// TIA Portal V21 export
FUNCTION_BLOCK "FB610"   // FB610, LAD
TITLE = FB610
{ S7_Optimized_Access := 'FALSE' }
AUTHOR : PRECISE
FAMILY : PRECISE
// CIP SYSTEM DRAIN
// stored: AutoNumber false, SetENOAutomatically false
   VAR_INPUT
      CycleEnable : Bool;
      CycleRunning : Bool;
      SecPulse : Bool;
      AlwaysTrue : Bool;
      SetTime : Int := 30;
      Loops : Int;
      DelayBetweenLoops : Int := 3;
   END_VAR
   VAR_OUTPUT
      Started : Bool;
      ParaOut : "SystemDrainOutputs";
      TimePv : DInt;
      StepStatus : String[60];
   END_VAR
   VAR_IN_OUT
      Over : Bool;
      OverTemp : Bool;
      Popup : Bool;
      PopupAck : Bool;
      PopUpSel : Bool;
   END_VAR
   VAR
      RE1 : Bool;
      "Timer" { S7_SetPoint := 'True'} : "FB101";
   END_VAR
   VAR_TEMP   // added for the SCL form of the ladder/FBD networks
      _w1 : Bool;
      _w2 : Bool;
      _w3 : Bool;
   END_VAR
BEGIN

REGION Network 1: SystemDrainStarted
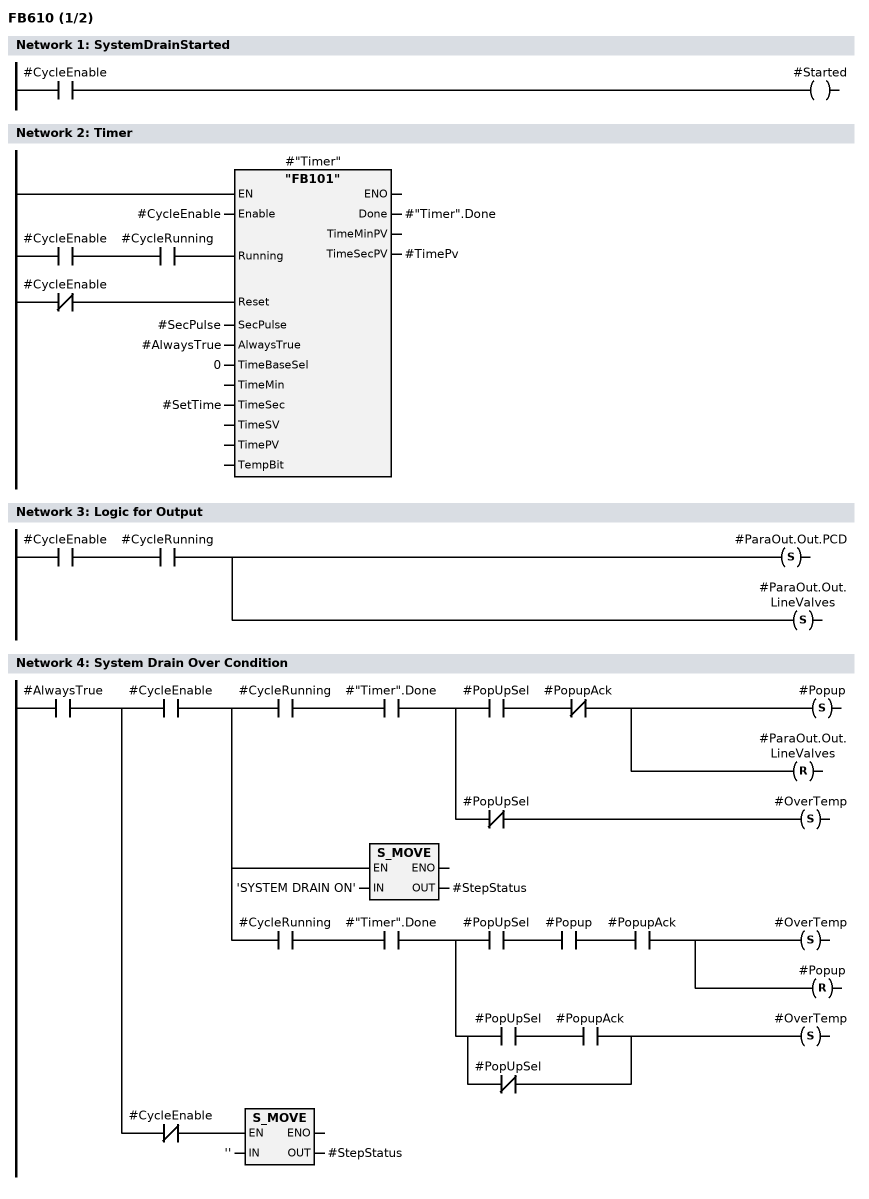
   RUNG wire#powerrail
      Contact( #CycleEnable )
      Coil( #Started )
   END_RUNG
   // the same network as SCL:
   #Started := #CycleEnable;
END_REGION

REGION Network 2: Timer
   RUNG wire#powerrail
      #"Timer"(Running := wire#w1, Reset := wire#w2, Enable := #CycleEnable, SecPulse := #SecPulse, AlwaysTrue := #AlwaysTrue, TimeBaseSel := 0, TimeMin :=, TimeSec := #SetTime, TimeSV :=, TimePV :=, TempBit :=, Done => #"Timer".Done, TimeMinPV =>, TimeSecPV => #TimePv)
   END_RUNG
   RUNG wire#powerrail
      Contact( #CycleEnable )
      Contact( #CycleRunning )
   END_RUNG wire#w1
   RUNG wire#powerrail
      I_Contact( #CycleEnable )
   END_RUNG wire#w2
   // the same network as SCL:
   #"Timer"(Enable := #CycleEnable,   // "FB101"
            Running := #CycleEnable AND #CycleRunning,
            Reset := NOT #CycleEnable,
            SecPulse := #SecPulse,
            AlwaysTrue := #AlwaysTrue,
            TimeBaseSel := 0,
            TimeSec := #SetTime,
            Done => #"Timer".Done,
            TimeSecPV => #TimePv);
END_REGION

REGION Network 3: Logic for Output
   RUNG wire#powerrail
      Contact( #CycleEnable )
      Contact( #CycleRunning )
      wire#w1
      S_Coil( #ParaOut.Out.PCD )
   END_RUNG
   RUNG wire#w1
      S_Coil( #ParaOut.Out.LineValves )
   END_RUNG
   // the same network as SCL:
   IF #CycleEnable AND #CycleRunning THEN
       #ParaOut.Out.PCD := TRUE;
       #ParaOut.Out.LineValves := TRUE;
   END_IF;
END_REGION

REGION Network 4: System Drain Over Condition
   RUNG wire#powerrail
      Contact( #AlwaysTrue )
      wire#w1
      Contact( #CycleEnable )
      wire#w2
      Contact( #CycleRunning )
      Contact( #"Timer".Done )
      wire#w3
      Contact( #PopUpSel )
      I_Contact( #PopupAck )
      wire#w4
      S_Coil( #Popup )
   END_RUNG
   RUNG wire#w4
      R_Coil( #ParaOut.Out.LineValves )
   END_RUNG
   RUNG wire#w3
      I_Contact( #PopUpSel )
      S_Coil( #OverTemp )
   END_RUNG
   RUNG wire#w2
      S_Move(in := 'SYSTEM DRAIN ON', out => #StepStatus)
   END_RUNG
   RUNG wire#w2
      Contact( #CycleRunning )
      Contact( #"Timer".Done )
      wire#w5
      Contact( #PopUpSel )
      Contact( #Popup )
      Contact( #PopupAck )
      wire#w6
      S_Coil( #OverTemp )
   END_RUNG
   RUNG wire#w6
      R_Coil( #Popup )
   END_RUNG
   RUNG wire#w5
      Contact( #PopUpSel )
      Contact( #PopupAck )
      wire#w7
      S_Coil( #OverTemp )
   END_RUNG
   RUNG wire#w5
      I_Contact( #PopUpSel )
   END_RUNG wire#w7
   RUNG wire#w1
      I_Contact( #CycleEnable )
      S_Move(in := '', out => #StepStatus)
   END_RUNG
   // the same network as SCL:
   #_w1 := #AlwaysTrue AND #CycleEnable;
   #_w2 := #_w1 AND #CycleRunning AND #"Timer".Done;
   IF #_w2 AND #PopUpSel AND NOT #PopupAck THEN
       #Popup := TRUE;
       #ParaOut.Out.LineValves := FALSE;
   END_IF;
   IF #_w2 AND NOT #PopUpSel THEN #OverTemp := TRUE; END_IF;
   IF #_w1 THEN #StepStatus := 'SYSTEM DRAIN ON'; END_IF;
   #_w3 := #_w1 AND #CycleRunning AND #"Timer".Done;
   IF #_w3 AND #PopUpSel AND #Popup AND #PopupAck THEN
       #OverTemp := TRUE;
       #Popup := FALSE;
   END_IF;
   IF #_w3 AND ((#PopUpSel AND #PopupAck) OR NOT #PopUpSel) THEN #OverTemp := TRUE; END_IF;
   IF #AlwaysTrue AND NOT #CycleEnable THEN #StepStatus := ''; END_IF;
END_REGION

REGION Network 5: System Drain Over
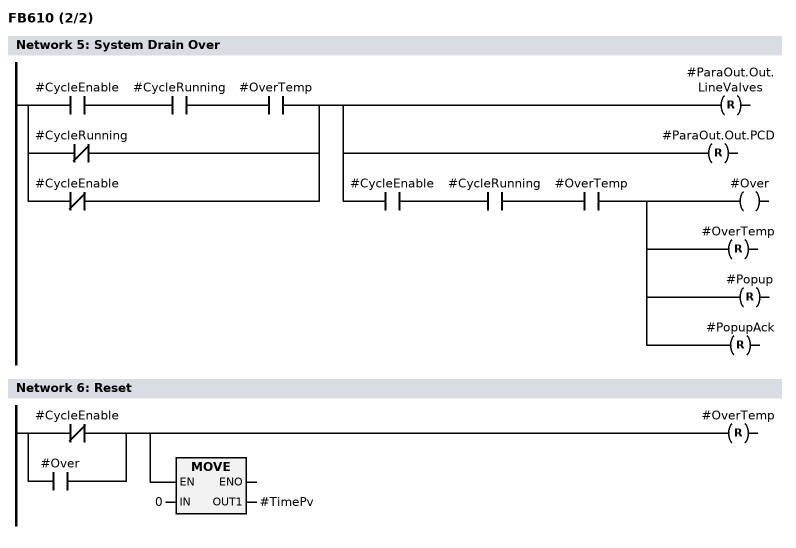
   RUNG wire#powerrail
      Contact( #CycleEnable )
      Contact( #CycleRunning )
      Contact( #OverTemp )
      wire#w1
      R_Coil( #ParaOut.Out.LineValves )
   END_RUNG
   RUNG wire#powerrail
      I_Contact( #CycleRunning )
   END_RUNG wire#w1
   RUNG wire#powerrail
      I_Contact( #CycleEnable )
   END_RUNG wire#w1
   RUNG wire#w1
      R_Coil( #ParaOut.Out.PCD )
   END_RUNG
   RUNG wire#w1
      Contact( #CycleEnable )
      Contact( #CycleRunning )
      Contact( #OverTemp )
      wire#w2
      Coil( #Over )
   END_RUNG
   RUNG wire#w2
      R_Coil( #OverTemp )
   END_RUNG
   RUNG wire#w2
      R_Coil( #Popup )
   END_RUNG
   RUNG wire#w2
      R_Coil( #PopupAck )
   END_RUNG
   // the same network as SCL:
   #_w1 := (#CycleEnable AND #CycleRunning AND #OverTemp) OR NOT #CycleRunning OR NOT #CycleEnable;
   IF #_w1 THEN
       #ParaOut.Out.LineValves := FALSE;
       #ParaOut.Out.PCD := FALSE;
   END_IF;
   #Over := #_w1 AND #CycleEnable AND #CycleRunning AND #OverTemp;
   IF #Over THEN
       #OverTemp := FALSE;
       #Popup := FALSE;
       #PopupAck := FALSE;
   END_IF;
END_REGION

REGION Network 6: Reset
   RUNG wire#powerrail
      I_Contact( #CycleEnable )
      wire#w1
      R_Coil( #OverTemp )
   END_RUNG
   RUNG wire#powerrail
      Contact( #Over )
   END_RUNG wire#w1
   RUNG wire#w1
      { S7_GenerateENO := "TRUE" } Move(in := 0, out1 => #TimePv)
   END_RUNG
   // the same network as SCL:
   IF NOT #CycleEnable OR #Over THEN
       #OverTemp := FALSE;
       #TimePv := 0;
   END_IF;
END_REGION
END_FUNCTION_BLOCK
